// Read Only Decorator for function blocks that impliment I_List interface
{attribute 'enable_dynamic_creation'}
FUNCTION_BLOCK FB_Read_Only_List EXTENDS FB_Collection IMPLEMENTS I_Read_Only_List
VAR_INPUT
	ipList : I_List;
END_VAR

(* Number of items in the collection*)
PROPERTY _Count : T_Capacity
GET
IF THIS^.NullReferenceException() THEN _Count := -1; RETURN; END_IF
_Count := THIS^.ipList._Count;
END_GET
END_PROPERTY

PROPERTY _Error_Status : ST_ERROR
GET
IF THIS^.NullReferenceException() THEN _Error_Status := THIS^.stError; RETURN; END_IF
THIS^.stError := THIS^.ipList._Error_Status;
_Error_Status := F_Error(THIS^.stError.bSTATUS, THIS^.stError.nCODE, THIS^.stError.sSOURCE);
END_GET
END_PROPERTY

(* Checks if collection is empty*)
PROPERTY _Is_Empty : BOOL
GET
IF THIS^.NullReferenceException() THEN _Is_Empty := TRUE; RETURN; END_IF
_Is_Empty := THIS^.ipList._Is_Empty;
END_GET
END_PROPERTY

(* DOES NOTHING - This is a read-only list *)
METHOD FINAL Clear
END_METHOD

(* Checks if item is contained in list *)
METHOD Contains : BOOL
VAR_INPUT
	Item : ANY; // Item to find in list
END_VAR
IF THIS^.NullReferenceException() THEN RETURN; END_IF
Contains := THIS^.ipList.Contains(Item);
END_METHOD

// Find the location of an item in list.
METHOD Find : I_Read_Only_List
VAR_INPUT
	Item 	: ANY; // Item to find in list
END_VAR
VAR_OUTPUT
	nIndex	: DINT; //Location of item in list 
	bSuccess : BOOL;
END_VAR
Find := THIS^;
IF THIS^.NullReferenceException() THEN nIndex := -1; RETURN; END_IF
THIS^.ipList.Find(Item, nIndex => nIndex, bSuccess => bSuccess);
END_METHOD

// Gets item from list at specified location without removing it
METHOD Get : I_Read_Only_List
VAR_INPUT
	Return_Item 	: ANY;  // Variable to store returned item
	nIndex 			: DINT; // Location of item
END_VAR
VAR_OUTPUT
	bSuccess : BOOL;
END_VAR
Get := THIS^;
IF THIS^.NullReferenceException() THEN RETURN; END_IF
THIS^.ipList.Get(Return_Item, nIndex, bSuccess => bSuccess);
END_METHOD

// Gets item at the front of the list 
METHOD Get_First : I_Read_Only_List
VAR_INPUT
	Return_Item 	: ANY; // Variable to store returned item
END_VAR
VAR_OUTPUT
	bSuccess : BOOL;
END_VAR
Get_First := THIS^;
IF THIS^.NullReferenceException() THEN RETURN; END_IF
THIS^.ipList.Get_First(Return_Item, bSuccess => bSuccess);
END_METHOD

// Gets item at the back of the list 
METHOD Get_Last : I_Read_Only_List
VAR_INPUT
	Return_Item 	: ANY; // Variable to store returned item
END_VAR
VAR_OUTPUT
	bSuccess : BOOL;
END_VAR
Get_Last := THIS^;
IF THIS^.NullReferenceException() THEN RETURN; END_IF
THIS^.ipList.Get_Last(Return_Item, bSuccess => bSuccess);
END_METHOD

// Returns item as a string, if type to string conversion is supported
METHOD Get_Value_As_String : I_Read_Only_List
VAR_INPUT
	nIndex	: DINT; // Location of item
END_VAR
VAR_OUTPUT
	sItem 	: T_MaxString; // Variable to store returned item
END_VAR
Get_Value_As_String := THIS^;
IF THIS^.NullReferenceException() THEN RETURN; END_IF
THIS^.ipList.Get_Value_As_String(nIndex, sItem => sItem);
END_METHOD

METHOD PROTECTED NullReferenceException : BOOL
NullReferenceException := THIS^.ipList = 0;
IF NOT NullReferenceException THEN RETURN; END_IF
THIS^.RaiseException(2000+GVL_CmpErrors.ERR_INVALID_REFERENCE, 'Null or Invalid Reference');
END_METHOD

END_FUNCTION_BLOCK

(* stored: Version 1.1.0.1, ProductVersion 3.1.4024.4
   POU FB_Read_Only_List: Id {6efe7c5c-a96b-4f7e-b188-16fc6ad6b70d}, SpecialFunc None
   Folder Exceptions: Id {acef49db-890d-409b-af55-d7f93b2291cb}
   Property _Count: Id {85c50e3d-78af-4a56-ab1f-bccf81c7a75a}
   Get Get: Id {6c8f504c-85ce-4ed9-aef0-83d5b593c0a2}
   Property _Error_Status: Id {f6286b31-d8e1-4195-bb1d-ab1cd49c0d81}
   Get Get: Id {a423cc1c-e241-4c5e-ac4a-5100b06f7459}
   Property _Is_Empty: Id {869a8107-32c9-4105-8aad-4c8aa73ae31a}
   Get Get: Id {cb3d1913-9d84-4879-a42e-6f522139cf44}
   Method Clear: Id {2d45307b-96ae-48e1-9b09-0f3dbe829bcc}
   Method Contains: Id {e5307dbf-b3b8-4998-b7a1-40f259c9f3e4}
   Method Find: Id {1440e5e6-ce20-46be-9150-fc7b20521a33}
   Method Get: Id {1d1eb80f-9dd8-4fbb-94f4-eae741a81e0d}
   Method Get_First: Id {626d40cd-4db1-4a6c-ba1a-fb37ae9e92c7}
   Method Get_Last: Id {3ee5f152-70c1-4cc0-92a8-24b33d586fc3}
   Method Get_Value_As_String: Id {698a4137-32d6-46eb-a34d-20a3b17fe57e}
   Method NullReferenceException: Id {75bd21d4-b795-41b2-bbbf-ed32d85d8aa0} *)
